Omron CX-Programmer project NewProject (CX-Programmer 9.61)

# PLC NewPLC1: CP1E N30

## Global symbols (name address type ; comment)
0.00 BOOL  ; PB1
100.00 BOOL  ; LAMP

## Program NewProgram1 (cyclic task 0)

### Section Section1

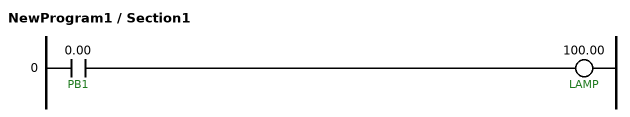
; rung 0
LD 0.00  ; PB1
OUT 100.00  ; LAMP
; rung 1
END(001)

### Section END
; rung 0
END(001)